% RSLogix 500 project I2P Hands-On 4 - Tanner.RSS, saved by version 10.00.00.00 %
PROJECT "UNTITLED"    % processor: Bul.1763 MicroLogix 1100 Series B %

PROGRAM FILES
  LAD 2   15 rungs

DATA FILES
  O0 OUTPUT  4 elements
  I1 INPUT  6 elements
  S2 STATUS  66 elements
  B3 BINARY  1 elements
  T4 TIMER  1 elements
  C5 COUNTER  1 elements
  R6 CONTROL  1 elements
  N7 INTEGER  1 elements
  F8 FLOAT  1 elements

LADDER 2
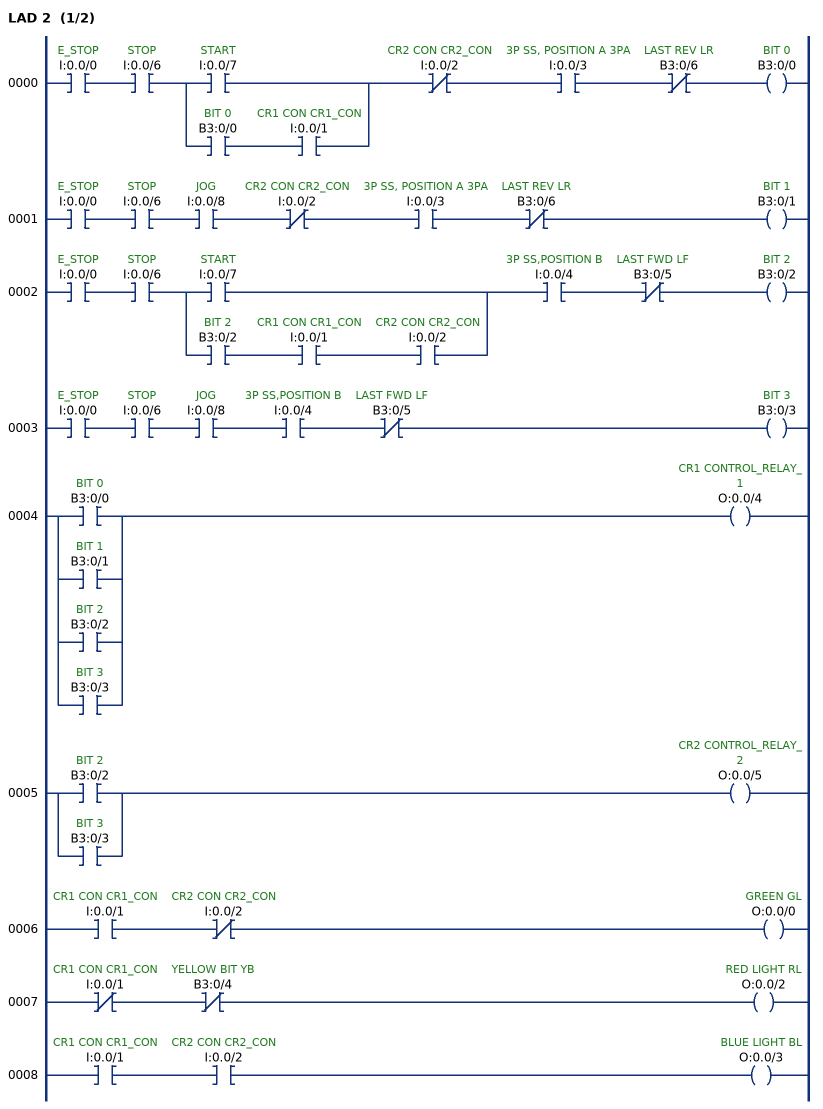
% Rung: 0 %
SOR XIC I:0.0/0 XIC I:0.0/6 BST XIC I:0.0/7 NXB XIC B3:0/0 XIC I:0.0/1 BND XIO I:0.0/2 XIC I:0.0/3 XIO B3:0/6 OTE B3:0/0 EOR
%   I:0.0/0  "E_STOP" %
%   I:0.0/6  "STOP" %
%   I:0.0/7  "START" %
%   B3:0/0  "BIT 0" %
%   I:0.0/1  CR1_CON  "CR1 CON" %
%   I:0.0/2  CR2_CON  "CR2 CON" %
%   I:0.0/3  3PA  "3P SS, POSITION A" %
%   B3:0/6  LR  "LAST REV" %
% Rung: 1 %
SOR XIC I:0.0/0 XIC I:0.0/6 XIC I:0.0/8 XIO I:0.0/2 XIC I:0.0/3 XIO B3:0/6 OTE B3:0/1 EOR
%   I:0.0/0  "E_STOP" %
%   I:0.0/6  "STOP" %
%   I:0.0/8  "JOG" %
%   I:0.0/2  CR2_CON  "CR2 CON" %
%   I:0.0/3  3PA  "3P SS, POSITION A" %
%   B3:0/6  LR  "LAST REV" %
%   B3:0/1  "BIT 1" %
% Rung: 2 %
SOR XIC I:0.0/0 XIC I:0.0/6 BST XIC I:0.0/7 NXB XIC B3:0/2 XIC I:0.0/1 XIC I:0.0/2 BND XIC I:0.0/4 XIO B3:0/5 OTE B3:0/2 EOR
%   I:0.0/0  "E_STOP" %
%   I:0.0/6  "STOP" %
%   I:0.0/7  "START" %
%   B3:0/2  "BIT 2" %
%   I:0.0/1  CR1_CON  "CR1 CON" %
%   I:0.0/2  CR2_CON  "CR2 CON" %
%   I:0.0/4  "3P SS,POSITION B" %
%   B3:0/5  LF  "LAST FWD" %
% Rung: 3 %
SOR XIC I:0.0/0 XIC I:0.0/6 XIC I:0.0/8 XIC I:0.0/4 XIO B3:0/5 OTE B3:0/3 EOR
%   I:0.0/0  "E_STOP" %
%   I:0.0/6  "STOP" %
%   I:0.0/8  "JOG" %
%   I:0.0/4  "3P SS,POSITION B" %
%   B3:0/5  LF  "LAST FWD" %
%   B3:0/3  "BIT 3" %
% Rung: 4 %
SOR BST BST BST XIC B3:0/0 NXB XIC B3:0/1 BND NXB XIC B3:0/2 BND NXB XIC B3:0/3 BND OTE O:0.0/4 EOR
%   B3:0/0  "BIT 0" %
%   B3:0/1  "BIT 1" %
%   B3:0/2  "BIT 2" %
%   B3:0/3  "BIT 3" %
%   O:0.0/4  CONTROL_RELAY_1  "CR1" %
% Rung: 5 %
SOR BST XIC B3:0/2 NXB XIC B3:0/3 BND OTE O:0.0/5 EOR
%   B3:0/2  "BIT 2" %
%   B3:0/3  "BIT 3" %
%   O:0.0/5  CONTROL_RELAY_2  "CR2" %
% Rung: 6 %
SOR XIC I:0.0/1 XIO I:0.0/2 OTE O:0.0/0 EOR
%   I:0.0/1  CR1_CON  "CR1 CON" %
%   I:0.0/2  CR2_CON  "CR2 CON" %
%   O:0.0/0  GL  "GREEN" %
% Rung: 7 %
SOR XIO I:0.0/1 XIO B3:0/4 OTE O:0.0/2 EOR
%   I:0.0/1  CR1_CON  "CR1 CON" %
%   B3:0/4  YB  "YELLOW BIT" %
%   O:0.0/2  RL  "RED LIGHT" %
% Rung: 8 %
SOR XIC I:0.0/1 XIC I:0.0/2 OTE O:0.0/3 EOR
%   I:0.0/1  CR1_CON  "CR1 CON" %
%   I:0.0/2  CR2_CON  "CR2 CON" %
%   O:0.0/3  BL  "BLUE LIGHT" %

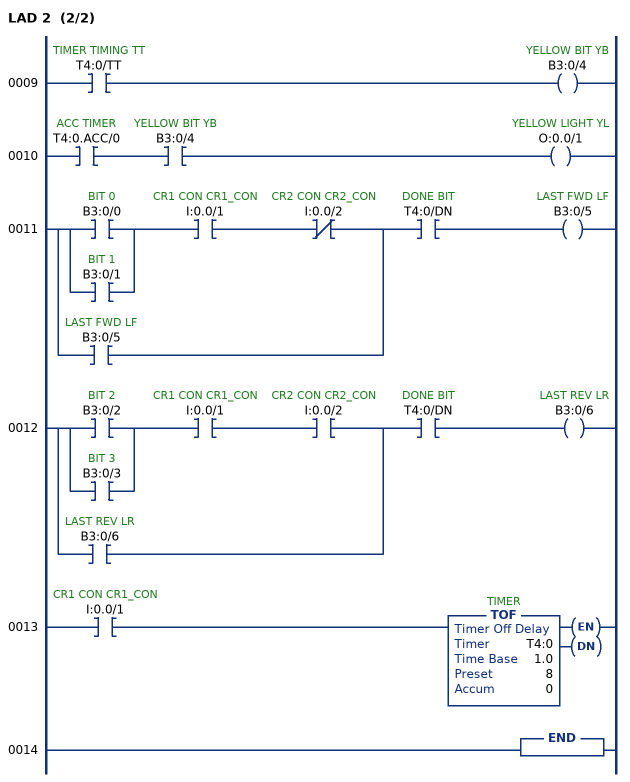
% Rung: 9 %
SOR XIC T4:0/TT OTE B3:0/4 EOR
%   T4:0/TT  TT  "TIMER TIMING" %
%   B3:0/4  YB  "YELLOW BIT" %
% Rung: 10 %
SOR XIC T4:0.ACC/0 XIC B3:0/4 OTE O:0.0/1 EOR
%   T4:0.ACC/0  "ACC TIMER" %
%   B3:0/4  YB  "YELLOW BIT" %
%   O:0.0/1  YL  "YELLOW LIGHT" %
% Rung: 11 %
SOR BST BST XIC B3:0/0 NXB XIC B3:0/1 BND XIC I:0.0/1 XIO I:0.0/2 NXB XIC B3:0/5 BND XIC T4:0/DN OTE B3:0/5 EOR
%   B3:0/0  "BIT 0" %
%   B3:0/1  "BIT 1" %
%   I:0.0/1  CR1_CON  "CR1 CON" %
%   I:0.0/2  CR2_CON  "CR2 CON" %
%   B3:0/5  LF  "LAST FWD" %
%   T4:0/DN  "DONE BIT" %
% Rung: 12 %
SOR BST BST XIC B3:0/2 NXB XIC B3:0/3 BND XIC I:0.0/1 XIC I:0.0/2 NXB XIC B3:0/6 BND XIC T4:0/DN OTE B3:0/6 EOR
%   B3:0/2  "BIT 2" %
%   B3:0/3  "BIT 3" %
%   I:0.0/1  CR1_CON  "CR1 CON" %
%   I:0.0/2  CR2_CON  "CR2 CON" %
%   B3:0/6  LR  "LAST REV" %
%   T4:0/DN  "DONE BIT" %
% Rung: 13 %
SOR XIC I:0.0/1 TOF T4:0 1.0 8 0 EOR
%   I:0.0/1  CR1_CON  "CR1 CON" %
%   T4:0  "TIMER" %
% Rung: 14 %
SOR END EOR

DATA TABLE (non-zero values as saved)
DATA T4
% .PRE .ACC %
% T4:0 % 8 0
